FUNCTION TryConvert_TIME_TO_DINT : BOOL
VAR_INPUT
	in : TIME;
	out : REFERENCE TO DINT;
END_VAR

IF in > DatatypeLimits.MAX_VALUE_OF_TIME_WHICH_CAN_BE_HELD_IN_A_DINT THEN
	RETURN;
END_IF

out := TIME_TO_DINT(in);
TryConvert_TIME_TO_DINT := TRUE;

END_FUNCTION

(* stored: Version 1.1.0.1, ProductVersion 3.1.4024.12
   POU TryConvert_TIME_TO_DINT: Id {49f285fe-dbb3-4a9b-876d-cb81a05566c8}, SpecialFunc None *)
